{attribute 'linkalways'} 
{attribute 'no_explicit_call' := 'This FB is a CLASS and must be accessed using methods or properties'}
{attribute 'enable_dynamic_creation'}
FUNCTION_BLOCK PUBLIC DeserializationFailedAlarm EXTENDS Alarm
VAR
	state : (CLEARED, RAISED);
	_reason : T_MAXSTRING;
END_VAR

PROPERTY Active : BOOL
GET
Active := state <> CLEARED;
END_GET
END_PROPERTY

METHOD PUBLIC Clear
_reason := '';
state := CLEARED;
END_METHOD

PROPERTY PUBLIC Message : T_MaxString
GET
Message := 'Deserialization failed';
END_GET
END_PROPERTY

METHOD PUBLIC Raise
VAR_INPUT
	Reason : T_MAXSTRING;
END_VAR
_reason := Reason;
state := RAISED;
END_METHOD

PROPERTY Reason : T_MaxString
GET
Reason := _reason;
END_GET
END_PROPERTY

END_FUNCTION_BLOCK

(* stored: Version 1.1.0.1, ProductVersion 3.1.4024.12
   POU DeserializationFailedAlarm: Id {c372a30f-c6a3-45ef-b720-6ac91004d584}, SpecialFunc None
   Property Active: Id {c6b994d7-412f-4d6a-bc1b-99506226df50}
   Get Get: Id {d0295560-17ac-47fc-bf19-83b33586945c}
   Method Clear: Id {d3b0e5a6-0425-4794-b362-0739af0aee5c}
   Property Message: Id {b47e6943-9ff4-4db9-9dc2-ccf830c0f517}
   Get Get: Id {8c60e1f4-530d-4060-ad96-eeed2a955569}
   Method Raise: Id {8b6e7914-ec13-4674-bb3e-5305ceef635e}
   Property Reason: Id {dde2c45e-eda3-430e-b3d8-a6bff36580f9}
   Get Get: Id {7700f3ca-38cf-4152-88eb-13864d7b9ab8} *)
